(* Logix 5000 project; controller jamiesFYP_PLC vendor 1 type 14 code 92 rev 35.12; software revision 35.01 *)

TASK MainTask (continuous, watchdog 500 ms) : MainProgram

MODULES
   Local : vendor 1 type 14 code 92 (ICP 0, rev 35.12)
      jamiesFYP_DCinput : vendor 1 type 7 code 2 (ICP 2, rev 3.1, Input RPI 20 ms)
      jamiesFYP_DCoutput : 1756-OB16D (ICP 1, rev 3.1, Output RPI 20 ms)
      jamiesFYP_Ethernet : 1756-EN2T (ICP 5, Ethernet 10.188.2.144, rev 11.1)
         GLW_LAB_LD_ROB01 : FANUC Robot R30iB Plus (Ethernet 10.188.2.186, rev 3.1, StandardDataDriven RPI 32 ms)
END_MODULES

VAR_GLOBAL   (* controller tags *)
   LDRobot_AtFullView : ALIAS FOR GLW_LAB_LD_ROB01:I1.Input[0].3;   // Robot at Fluke Full View
   LDRobot_AtHomePos : ALIAS FOR GLW_LAB_LD_ROB01:I1.Input[0].0;   // Robot at Home Pos
   LDRobot_AtPos1 : ALIAS FOR GLW_LAB_LD_ROB01:I1.Input[0].1;   // Robot at Fluke Pos 1
   LDRobot_AtPos2 : ALIAS FOR GLW_LAB_LD_ROB01:I1.Input[0].2;   // Robot at Fluke Pos 2
   LDRobot_CycleComplete : ALIAS FOR GLW_LAB_LD_ROB01:I1.Input[0].4;   // Robot Cycle Complete
   LDRobot_Reset : ALIAS FOR GLW_LAB_LD_ROB01:O1.Output[0].1;   // Reset Signal
   LDRobot_StartCycle : ALIAS FOR GLW_LAB_LD_ROB01:O1.Output[0].0;   // Start Signal to Robot
   LDRobot_TestCompleteAck : ALIAS FOR GLW_LAB_LD_ROB01:O1.Output[0].2;   // Awknowledge Cycle Complete
END_VAR

PROGRAM MainProgram   (* main routine MainRoutine *)

ROUTINE MainRoutine   (* ladder *)
END_ROUTINE
END_PROGRAM
